TYPE Interlock :
STRUCT
	interlockSetting : InterlockSetting;
	interlockState : InterlockState;
	Interlock_Return_Message :T_MaxString;  (*plc에서 특정 Trig를 True로 바꾸면 UI에서는 이 메시지를 Popup ??   *)
END_STRUCT
END_TYPE

(* stored: Version 1.1.0.1, ProductVersion 3.1.4026.11
   DUT Interlock: Id {cd6f6425-6313-4e47-b815-d7dccd73d4bd} *)
